INTERFACE IAnalogValue16BitConverter EXTENDS Core.IObject

METHOD ConvertAnalogValueToRawValue : WORD
VAR_INPUT
	analogValue : LREAL;
END_VAR
END_METHOD

METHOD ConvertRawValueToAnalogValue : LREAL
VAR_INPUT
	rawValue : WORD;
END_VAR
END_METHOD

END_INTERFACE

(* stored: Version 1.1.0.1
   Itf IAnalogValue16BitConverter: Id {996c28a6-ed43-435b-bd2d-4a48e125454f}
   Method ConvertAnalogValueToRawValue: Id {7b9f8ba6-8d64-4125-89ee-b6b6b6ab7033}
   Method ConvertRawValueToAnalogValue: Id {8ee92332-8449-42df-aea2-819ba3290c45} *)
